// TIA Portal V20 export
VAR_GLOBAL   // PLC tag table "Unit1Em2"
   "BA010AZCRBK01.02" AT %I1000.2 : Bool;   // UW SUPPORT UNIT TRANSFER BACKWARD
   "BA010AZCRBK01.03" AT %I1000.3 : Bool;   // ELECTRODE SHAFT SUPPORTER DOWN
   "BA010AZCRBK01.05" AT %I1000.5 : Bool;   // ELECTRODE FIX LEFT TOP PRESSURE SWITCH
   "BA010AZCRBK01.12" AT %I1001.2 : Bool;   // UW SUPPORT UNIT TRANSFER FORWARD
   "BA010AZCRBK01.13" AT %I1001.3 : Bool;   // ELECTRODE SHAFT SUPPORTER UP
   "BA010AZCRBK01.15" AT %I1001.5 : Bool;   // ELECTRODE FIX LEFT BTM PRESSURE SWITCH
   "BA010AZCRPM01.10" AT %Q2001.0 : Bool;   // UNWINDER SUPPORT UNIT TRANSFER FORWARD
   "BA010AZCRPM01.11" AT %Q2001.1 : Bool;   // UNWINDER SUPPORT UNIT TRANSFER BACKWARD
   "BA010AZCRPM01.12" AT %Q2001.2 : Bool;   // ELECTRODE SHAFT SUPPORTER UP
   "BA010AZCRPM01.13" AT %Q2001.3 : Bool;   // ELECTRODE SHAFT SUPPORTER DOWN
   "BA010AZCRBK02.00" AT %I1004.0 : Bool;   // ELECTRODE FIX RIGHT TOP BACKWARD
   "BA010AZCRBK02.01" AT %I1004.1 : Bool;   // ELECTRODE FIX RIGHT TOP FORWARD
   "BA010AZCRBK02.02" AT %I1004.2 : Bool;   // ELECTRODE FIX RIGHT BTM BACKWARD
   "BA010AZCRBK02.03" AT %I1004.3 : Bool;   // ELECTRODE FIX RIGHT BTM FORWARD
   "BA010AZCRBK02.04" AT %I1004.4 : Bool;   // ELECTRODE FIX RIGHT TOP PRESSURE SWITCH
   "BA010AZCRBK02.05" AT %I1004.5 : Bool;   // ELECTRODE FIX RIGHT BTM PRESSURE SWITCH
   "BA010AZCRBK02.06" AT %I1004.6 : Bool;   // ELECTRODE CUTTER BACKWARD
   "BA010AZCRPM02.01" AT %Q2004.1 : Bool;   // UNWINDER SPLICER RIGHT ELECTRODE FIX RIGHT TOP BACKWARD
   "BA010AZCRPM02.02" AT %Q2004.2 : Bool;   // UNWINDER SPLICER RIGHT ELECTRODE FIX RIGHT BTM FORWARD
   "BA010AZCRPM02.03" AT %Q2004.3 : Bool;   // UNWINDER SPLICER RIGHT ELECTRODE FIX RIGHT BTM BACKWARD
   "BA010AZCRPM02.04" AT %Q2004.4 : Bool;   // UNWINDER SPLICER RIGHT CUTTER FORWARD
   "BA010AZCRPM02.05" AT %Q2004.5 : Bool;   // UNWINDER SPLICER RIGHT CUTTER BACKWARD
   "BA010AZCRPM02.06" AT %Q2004.6 : Bool;   // UNWINDER SPLICER LEFT ELECTRODE FIX LEFT TOP FORWARD
   "BA010AZCRPM02.07" AT %Q2004.7 : Bool;   // UNWINDER SPLICER LEFT ELECTRODE FIX LEFT TOP BACKWARD
   "BA010AZCRPM02.10" AT %Q2005.0 : Bool;   // UNWINDER SPLICER LEFT ELECTRODE FIX LEFT BTM FORWARD
   "BA010AZCRPM02.11" AT %Q2005.1 : Bool;   // UNWINDER SPLICER LEFT ELECTRODE FIX LEFT BTM BACKWARD
   "BA010AZCRPM02.12" AT %Q2005.2 : Bool;   // UNWINDER SPLICER LEFT ELECTRODE FIX LEFT TOP DOWN
   "BA010AZCRPM02.13" AT %Q2005.3 : Bool;   // UNWINDER SPLICER LEFT ELECTRODE FIX LEFT TOP UP
   "BA010AZCRPM02.14" AT %Q2005.4 : Bool;   // UNWINDER SPLICER LEFT ELECTRODE FIX LEFT BTM UP
   "BA010AZCRPM02.15" AT %Q2005.5 : Bool;   // UNWINDER SPLICER LEFT ELECTRODE FIX LEFT BTM DOWN
   "BA010AZCRBK03.00" AT %I1008.0 : Bool;   // ELECTRODE FIX LEFT TOP BACKWARD
   "BA010AZCRBK03.01" AT %I1008.1 : Bool;   // UNWINDER STOPPER BACKWARD
   "BA010AZCRBK03.02" AT %I1008.2 : Bool;   // ELECTRODE FIX LEFT BTM BACKWARD
   "BA010AZCRBK03.04" AT %I1008.4 : Bool;   // ELECTRODE FIX LEFT TOP UP
   "BA010AZCRBK03.05" AT %I1008.5 : Bool;   // FRAME COVER BACKWARD
   "BA010AZCRBK03.06" AT %I1008.6 : Bool;   // ELECTRODE FIX LEFT BTM DOWN
   "BA010AZCRBK03.10" AT %I1009.0 : Bool;   // ELECTRODE FIX LEFT TOP FORWARD
   "BA010AZCRBK03.11" AT %I1009.1 : Bool;   // UNWINDER STOPPER FORWARD
   "BA010AZCRBK03.12" AT %I1009.2 : Bool;   // ELECTRODE FIX LEFT BTM FORWARD
   "BA010AZCRBK03.14" AT %I1009.4 : Bool;   // ELECTRODE FIX LEFT TOP DOWN
   "BA010AZCRBK03.15" AT %I1009.5 : Bool;   // FRAME COVER FORWARD
   "BA010AZCRBK03.16" AT %I1009.6 : Bool;   // ELECTRODE FIX LEFT BTM UP
   "BA010AZCRPM03.00" AT %Q2008.0 : Bool;   // UNWINDER SPLICER HOLDER SPLICING LEFT MODULE MOVER FORWARD
   "BA010AZCRPM03.01" AT %Q2008.1 : Bool;   // UNWINDER SPLICER HOLDER SPLICING LEFT MODULE MOVER BACKWARD
   "BA010AZCRPM03.02" AT %Q2008.2 : Bool;   // UNWINDER SPLICER HOLDER SPLICING RIGHT MODULE MOVER FORWARD
   "BA010AZCRPM03.03" AT %Q2008.3 : Bool;   // UNWINDER SPLICER HOLDER SPLICING RIGHT MODULE MOVER BACKWARD
   "BA010AZCRPM03.04" AT %Q2008.4 : Bool;   // UNWINDER SPLICER HOLDER ELECTRODE LEFT HOLDER MODULE MOVER FORWARD
   "BA010AZCRPM03.05" AT %Q2008.5 : Bool;   // UNWINDER SPLICER HOLDER ELECTRODE LEFT HOLDER MODULE MOVER BACKWARD
   "BA010AZCRPM03.06" AT %Q2008.6 : Bool;   // UNWINDER SPLICER HOLDER ELECTRODE RIGHT HOLDER MODULE MOVER FORWARD
   "BA010AZCRPM03.07" AT %Q2008.7 : Bool;   // UNWINDER SPLICER HOLDER ELECTRODE RIGHT HOLDER MODULE MOVER BACKWARD
   "BA010AZCRPM03.10" AT %Q2009.0 : Bool;   // UNWINDER SPLICER TAPE LOADING TURN ROTATE
   "BA010AZCRPM03.11" AT %Q2009.1 : Bool;   // UNWINDER SPLICER TAPE LOADING TURN HOME
   "BA010AZCRPM03.12" AT %Q2009.2 : Bool;   // UNWINDER SPLICER TAPE ATTACH UNIT FORWARD
   "BA010AZCRPM03.13" AT %Q2009.3 : Bool;   // UNWINDER SPLICER TAPE ATTACH UNIT BACKWARD
   "BA010AZCRBK04.00" AT %I1012.0 : Bool;   // SPLICING L-MODULE MOVER BACKWARD
   "BA010AZCRBK04.01" AT %I1012.1 : Bool;   // SPLICING R-MODULE MOVER BACKWARD
   "BA010AZCRBK04.02" AT %I1012.2 : Bool;   // ELECTRODE L-HOLDER MOVER FORWARD
   "BA010AZCRBK04.03" AT %I1012.3 : Bool;   // ELECTRODE R-HOLDER MOVER FORWARD
   "BA010AZCRBK04.04" AT %I1012.4 : Bool;   // TAPE LOADING TURN HOMING
   "BA010AZCRBK04.05" AT %I1012.5 : Bool;   // TAPE ATTACH UNIT BACKWARD
   "BA010AZCRBK04.06" AT %I1012.6 : Bool;   // TAPING VACUUM PRESSURE SWITCH
   "BA010AZCRBK04.10" AT %I1013.0 : Bool;   // SPLICING L-MODULE MOVER FORWARD
   "BA010AZCRBK04.11" AT %I1013.1 : Bool;   // SPLICING R-MODULE MOVER FORWARD
   "BA010AZCRBK04.12" AT %I1013.2 : Bool;   // ELECTRODE L-HOLDER MOVER BACKWARD
   "BA010AZCRBK04.13" AT %I1013.3 : Bool;   // ELECTRODE R-HOLDER MOVER BACKWARD
   "BA010AZCRBK04.14" AT %I1013.4 : Bool;   // TAPE LOADING TURN ROTATE
   "BA010AZCRBK04.15" AT %I1013.5 : Bool;   // TAPE ATTACH UNIT FORWARD
   "BA010AZCRPM04.00" AT %Q2012.0 : Bool;   // UNWINDER STOPPER FORWARD
   "BA010AZCRPM04.01" AT %Q2012.1 : Bool;   // UNWINDER STOPPER BACKWARD
   "BA010AZCRPM04.16" AT %Q2013.6 : Bool;   // FRAME COVER FORWARD
   "BA010AZCRPM04.17" AT %Q2013.7 : Bool;   // FRAME COVER BACKWARD
   "BA010AZCRBK08.00" AT %Q2100.0 : Bool;   // UW ELECTRODE FIX LEFT TOP V/C ON
   "BA010AZCRBK08.01" AT %Q2100.1 : Bool;   // UW ELECTRODE FIX LEFT TOP V/C OFF
   "BA010AZCRBK08.02" AT %Q2100.2 : Bool;   // UW ELECTRODE FIX LEFT BTM V/C ON
   "BA010AZCRBK08.03" AT %Q2100.3 : Bool;   // UW ELECTRODE FIX LEFT BTM V/C OFF
   "BA010AZCRBK08.04" AT %Q2100.4 : Bool;   // UW ELECTRODE FIX RIGHT TOP V/C ON
   "BA010AZCRBK08.05" AT %Q2100.5 : Bool;   // UW ELECTRODE FIX RIGHT TOP V/C OFF
   "BA010AZCRBK08.06" AT %Q2100.6 : Bool;   // UW ELECTRODE FIX RIGHT BTM V/C ON
   "BA010AZCRBK08.07" AT %Q2100.7 : Bool;   // UW ELECTRODE FIX RIGHT BTM V/C OFF
   "BA010AZCRBK10.00" AT %Q2108.0 : Bool;   // UW TAPE ATTACH V/C ON
   "BA010AZCRBK10.01" AT %Q2108.1 : Bool;   // UW TAPE ATTACH V/C OFF
   "BA010AZCRBK10.02" AT %Q2108.2 : Bool;   // CART DETECT CHECK LAMP
   "BA010AZCRBK02.07" AT %I1004.7 : Bool;   // ELECTRODE CUTTER FORWARD
   "BA010AZCRPM02.00" AT %Q2004.0 : Bool;   // UNWINDER SPLICER RIGHT ELECTRODE FIX RIGHT TOP FORWARD
END_VAR
VAR_GLOBAL CONSTANT   // user constants
   U1EM2_JOB01 : DInt := 1;
   U1EM2_JOB02 : DInt := 2;
   U1EM2_JOB03 : DInt := 3;
   U1EM2_JOB04 : DInt := 4;
   U1EM2_JOB05 : DInt := 5;
   U1EM2_JOB06 : DInt := 6;
   U1EM2_JOB07 : DInt := 7;
   U1EM2_JOB08 : DInt := 8;
   U1EM2_JOB09 : DInt := 9;
   U1EM2_JOB10 : DInt := 10;
   U1EM2_JOB11 : DInt := 11;
   U1EM2_JOB12 : DInt := 12;
   U1EM2_JOB13 : DInt := 13;
   U1EM2_JOB14 : DInt := 14;
   U1EM2_JOB15 : DInt := 15;
   U1EM2_JOB16 : DInt := 16;
   U1EM2_JOB17 : DInt := 17;
   U1EM2_JOB18 : DInt := 18;
   U1EM2_JOB19 : DInt := 19;
   U1EM2_JOB20 : DInt := 20;
   U1EM2_JOB21 : DInt := 21;
   U1EM2_JOB22 : DInt := 22;
   U1EM2_JOB23 : DInt := 23;
   U1EM2_JOB24 : DInt := 24;
   U1EM2_JOB25 : DInt := 25;
   U1EM2_JOB26 : DInt := 26;
   U1EM2_JOB27 : DInt := 27;
   U1EM2_JOB28 : DInt := 28;
   U1EM2_JOB29 : DInt := 29;
   U1EM2_JOB30 : DInt := 30;
   U1EM2_JOB31 : DInt := 31;
   U1EM2_JOB32 : DInt := 32;
   U1EM2_JOB33 : DInt := 33;
   U1EM2_JOB34 : DInt := 34;
   U1EM2_JOB35 : DInt := 35;
   U1EM2_JOB36 : DInt := 36;
   U1EM2_JOB37 : DInt := 37;
   U1EM2_JOB38 : DInt := 38;
   U1EM2_JOB39 : DInt := 39;
   U1EM2_JOB40 : DInt := 40;
   U1EM2_JOB41 : DInt := 41;
   U1EM2_JOB42 : DInt := 42;
   U1EM2_JOB43 : DInt := 43;
   U1EM2_JOB44 : DInt := 44;
   U1EM2_JOB45 : DInt := 45;
   U1EM2_JOB46 : DInt := 46;
   U1EM2_JOB47 : DInt := 47;
   U1EM2_JOB48 : DInt := 48;
   U1EM2_JOB49 : DInt := 49;
   U1EM2_JOB50 : DInt := 50;
END_VAR
